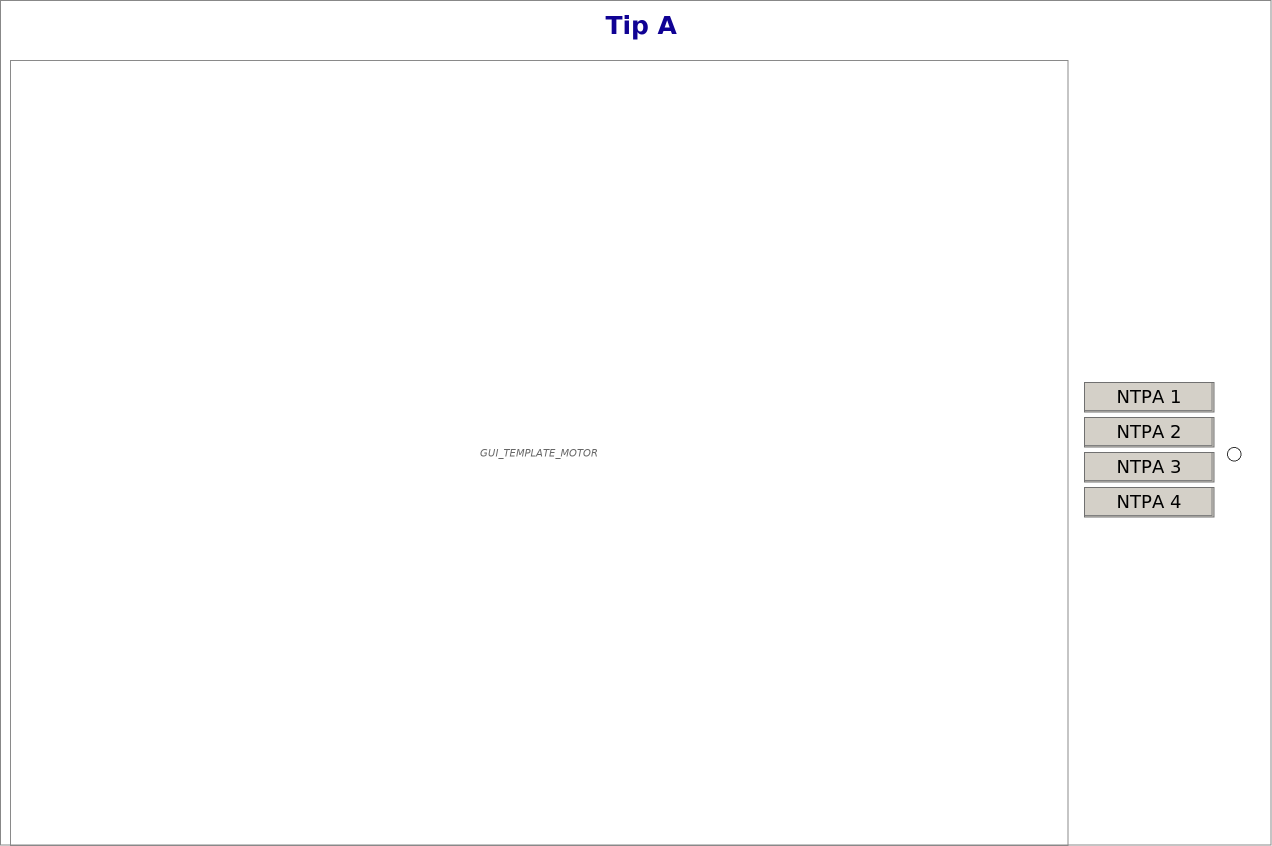
VISUALIZATION VISU_HMI_TIP_A  // 1272x846
    Group (10,10 1262x836)
        Label (532,0 199x30), "Tip A"
        Frame (0,50 1058x786)
            shows GUI_TEMPLATE_MOTOR(m_Instance := MAIN.nott_ics.TipTilt.ptrTipActuatorsA[MAIN.nott_ics.TipTilt.guiTipActuatorsAIndex]^)
        RadioButton (1215,374 47x140), variable: MAIN.nott_ics.TipTilt.guiTipActuatorsAIndex-1
            Areas[0]: Text=Radiobutton
            Areas[1]: Text=Radiobutton
        Button (1074,372 130x30), "NTPA 1"
            OnMouseClick: execute { MAIN.nott_ics.TipTilt.guiTipActuatorsAIndex := 1; }
        Button (1074,407 130x30), "NTPA 2"
            OnMouseClick: execute { MAIN.nott_ics.TipTilt.guiTipActuatorsAIndex := 2; }
        Button (1074,442 130x30), "NTPA 3"
            OnMouseClick: execute { MAIN.nott_ics.TipTilt.guiTipActuatorsAIndex := 3; }
        Button (1074,477 130x30), "NTPA 4"
            OnMouseClick: execute { MAIN.nott_ics.TipTilt.guiTipActuatorsAIndex := 4; }
END_VISUALIZATION

(* stored: Version 1.1.0.1, ProductVersion 3.1.4024.15
   Visu VISU_HMI_TIP_A: Id {c53dcc67-0a19-47ef-8cb3-c5834aaae248} *)
